// Core §3.15.1a — neutral byte-transport state (non-blocking, observed over scans).
{attribute 'qualified_only'}
TYPE E_ByteChannelState : (CLOSED := 0, OPENING := 1, OPEN := 2, FAULT := 3) DINT;
END_TYPE

(* stored: Version 1.1.0.1, ProductVersion 3.1.4024.12
   DUT E_ByteChannelState: Id {73341db2-cede-4369-b09b-e606db469286} *)
